FUNCTION projArray0 : DINT
VAR_INPUT
	arr: ARRAY[0..3] OF DINT;
	idx: DINT;
END_VAR

projArray0 := arr[normProjIdx(idx, 4)];

END_FUNCTION

(* stored: Version 1.1.0.1, ProductVersion 3.1.4022.18
   POU projArray0: Id {a9c41957-ce40-490b-9977-52db6538d385}, SpecialFunc None *)
